TYPE FsT_Size : UXINT; END_TYPE

(* stored: Version 1.1.0.1, ProductVersion 3.1.4024.4
   DUT FsT_Size: Id {4b57b667-d024-4dac-8788-462811423595} *)
